PROGRAM MAIN
VAR
	aOneArray : ARRAY[1..5] OF INT := [4, 20, 30, 40, 50];
	nOneInt : INT;
END_VAR

aOneArray[1] := 42;
nOneInt := aOneArray[1] + aOneArray[4];

END_PROGRAM

(* stored: Version 1.1.0.1, ProductVersion 3.1.4024.11
   POU MAIN: Id {c97b8ca2-ef16-4241-894c-346f57c19328}, SpecialFunc None *)
